ABB RobotStudio station: 23.rsstn

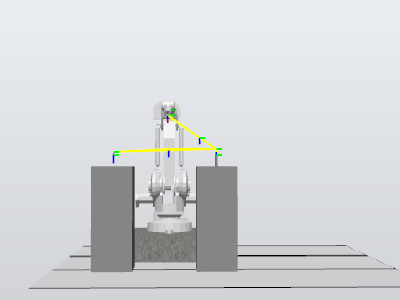
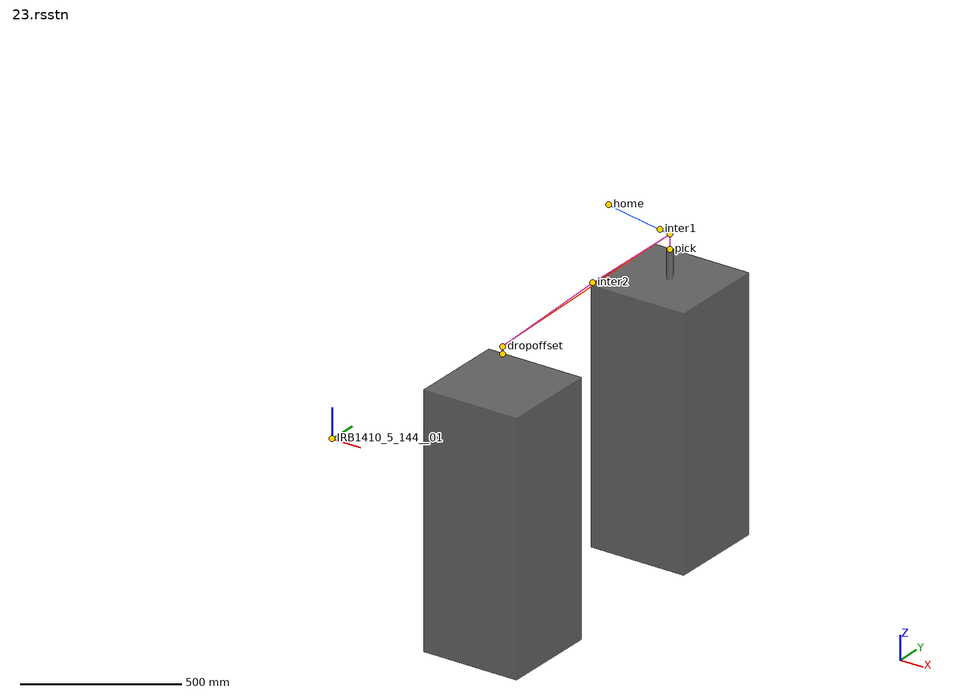
[picture v1: parts stored in the station drawn from their meshes, with robot base, taught points and paths (robot models come from the ABB library and are not in the file)]
Station Station (saved by RobotStudio 22.3.10141.1)
Controller Controller10, task T_ROB1: task frame (RAPID world) sits at (0, 0, 247) mm in the station
Controller Controller10
  mechanical unit ROB_1: IRB1410_5_144__01, 6 joints, base frame (0, 0, 0) mm
Layout (positions relative to the parent item):
  - Concrete [part, from Dispencing\Concrete.rslib]
  - IRB1410_5_144__01 [mechanism, from Robots\IRB1410_5_144_G_01.rslib] at (0, 0, 247) mm; joint values [0, 0, 0, 0, 0.5236, 0] (rad or m)
  - Part_1 [part] at (800, 250, 0) mm, size 350 x 350 x 900 mm
  - Part_2 [part] at (800, -650, 0) mm, size 350 x 350 x 900 mm
  - Part_3 [part] at (975, 425, 900) mm, size 24 x 23.9 x 100 mm
  - Part_4 [part] at (975, -475, 900) mm, size 24 x 23.9 x 100 mm
  - SmartComponent_1 [smart component] at (943.61, 0, 1399.5) mm, rotated rx -180 ry 60 rz -180 deg
      signals: DI close
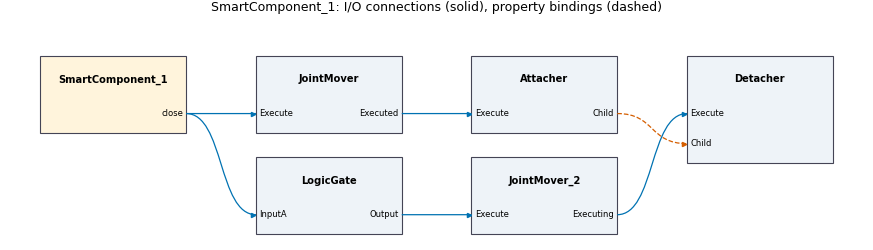
      connections:
        JointMover.Executed -> Attacher.Execute
        JointMover_2.Executing -> Detacher.Execute
        SmartComponent_1.close -> JointMover.Execute
        SmartComponent_1.close -> LogicGate.InputA
        LogicGate.Output -> JointMover_2.Execute
        Attacher.Child => Detacher.Child
    - LogicGate [smart component, from Components\LogicGate.rslib]
        properties: Operator=NOT; Delay=0
    - Detacher [smart component, from Components\Detacher.rslib]
        properties: Child=Part_3; KeepPosition=true
    - Attacher [smart component, from Components\Attacher.rslib]
        properties: Parent=Smart_Gripper_Servo_Fingers; Flange=0; Child=Part_3; Mount=false; Offset=[0 0 0]; Orientation=[0 0 0]
    - JointMover [smart component, from Components\JointMover.rslib]
        properties: Mechanism=Smart_Gripper_Servo_Fingers; Relative=false; Duration=0; J1=0.023
    - JointMover_2 [smart component, from Components\JointMover.rslib]
        properties: Mechanism=Smart_Gripper_Servo_Fingers; Relative=false; Duration=0; J1=0.025
    - Smart_Gripper_Servo_Fingers [mechanism, from Tools\ABB_Smart_Gripper_Servo_Fingers.rslib] at (0, 0, 0) mm; joint values [0.025] (rad or m)
Attachment: SmartComponent_1 is attached to IRB1410_5_144__01 / Link6
Station logic (signal -> signal, property => property):
  Controller10.att -> SmartComponent_1.close
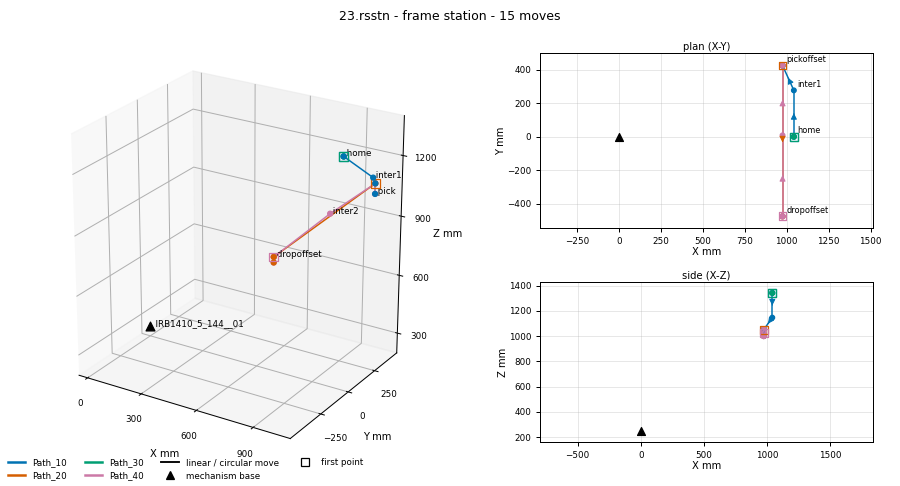
[picture p0: tool path of 23.rsstn in frame station, 15 of 15 moves have a stored position in this frame; points joined in program order, loops and branches not executed]
Targets, tools, work objects and paths stored in the station, written as RAPID:
! task T_ROB1
MODULE CalibData
  PERS tooldata Servo:=[TRUE,[[0,0,114.2],[1,0,0,0]],[0.215,[8.7,12.3,49.2],[1,0,0,0],0.00021,0.00024,0.00009]];
ENDMODULE

! task T_ROB1
MODULE Module1
  CONST robtarget home:=[[1042.512260434,0,1095.4],[0.5,0,0.866025404,0],[0,0,0,0],[9E+09,9E+09,9E+09,9E+09,9E+09,9E+09]];
  CONST robtarget inter1:=[[1042.512018861,276.810200353,899.723823207],[0.324673417,-0.000000015,0.945826185,0.000000003],[0,-1,0,0],[9E+09,9E+09,9E+09,9E+09,9E+09,9E+09]];
  CONST robtarget pick:=[[974.999996779,424.999984661,753.000009041],[-0.000000006,0,1,-0.000000003],[0,-1,0,0],[9E+09,9E+09,9E+09,9E+09,9E+09,9E+09]];
  CONST robtarget pickoffset:=[[974.999974457,424.999905774,805.223476216],[0.000000096,0.000000089,1,0.000000042],[0,0,0,0],[9E+09,9E+09,9E+09,9E+09,9E+09,9E+09]];
  CONST robtarget inter2:=[[974.999978527,8.314954096,805.22351945],[0.000000097,0.000000089,1,0.000000054],[0,0,0,0],[9E+09,9E+09,9E+09,9E+09,9E+09,9E+09]];
  CONST robtarget drop:=[[975.000039554,-474.999675513,752.999711764],[0.000000087,0.000000086,1,0.000000058],[-1,0,-1,0],[9E+09,9E+09,9E+09,9E+09,9E+09,9E+09]];
  CONST robtarget dropoffset:=[[974.999985439,-474.999685104,779.116918948],[0.00000008,0.000000082,1,0.000000062],[-1,0,-1,0],[9E+09,9E+09,9E+09,9E+09,9E+09,9E+09]];
  PROC Path_10()
    MoveL home,v1000,z100,Servo\WObj:=wobj0;
    MoveL inter1,v1000,z100,Servo\WObj:=wobj0;
    MoveL pickoffset,v1000,z100,Servo\WObj:=wobj0;
    MoveL pick,v1000,z100,Servo\WObj:=wobj0;
    WaitTime 1;
    SetDO att,1;
  ENDPROC
  PROC Path_20()
    MoveL pickoffset,v1000,z100,Servo\WObj:=wobj0;
    MoveL dropoffset,v1000,z100,Servo\WObj:=wobj0;
    MoveL drop,v1000,z100,Servo\WObj:=wobj0;
    WaitTime 1;
    SetDO att,0;
  ENDPROC
  PROC Path_30()
    Path_10;
    Path_20;
    MoveL home,v1000,z100,Servo\WObj:=wobj0;
    Path_40;
    MoveL home,v1000,z100,Servo\WObj:=wobj0;
  ENDPROC
  PROC Path_40()
    MoveL dropoffset,v1000,z100,Servo\WObj:=wobj0;
    MoveL drop,v1000,z100,Servo\WObj:=wobj0;
    WaitTime 1;
    SetDO att,1;
    MoveL dropoffset,v1000,z100,Servo\WObj:=wobj0;
    MoveL inter2,v1000,z100,Servo\WObj:=wobj0;
    MoveL pickoffset,v1000,z100,Servo\WObj:=wobj0;
    MoveL pick,v1000,z100,Servo\WObj:=wobj0;
    WaitTime 1;
    SetDO att,0;
  ENDPROC
  PROC main()
  ENDPROC
ENDMODULE

